FUNCTION_BLOCK BOXCOLOR_TO_COLOR (* Enum to Color *)
  (* Standard: 61499-2 *)
  (* Version 0.3, 2009-09-15, JHC, Holobloc Inc, Changed transition priorities. *)
  (* Version 0.2, 2003-12-04, JHC, Rockwell Automation, Renamed for better indexing. *)
  (* Version 0.1, 2002-11-05, JHC, Rockwell Automation, Corrected missing ST element in Algorithm REQ. *)
  (* Version 0.0, 2000-05-30, JHC, Rockwell Automation *)
  (* Compiler header: package fb.rt.dasdA1.A2.Box; *)
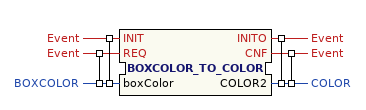
  EVENT_INPUT
    INIT WITH boxColor; (* Initialization Request *)
    REQ WITH boxColor; (* Normal Execution Request *)
  END_EVENT
  EVENT_OUTPUT
    INITO WITH COLOR2; (* Initialization Confirm *)
    CNF WITH COLOR2; (* Execution Confirmation *)
  END_EVENT
  VAR_INPUT
    boxColor : BOXCOLOR; (* BOXCOLOR ENUM *)
  END_VAR
  VAR_OUTPUT
    COLOR2 : COLOR; (* Color *)
  END_VAR
  VAR
    C2 : COLOR := COLOR#YELLOW;
    C3 : COLOR := COLOR#BLUE;
    C1 : COLOR := COLOR#RED;
  END_VAR
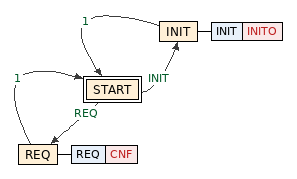
  EC_STATES
    START; (* Initial State *)
    INIT : INIT -> INITO; (* Initialization *)
    REQ : REQ -> CNF; (* Normal execution *)
  END_STATES
  EC_TRANSITIONS
    INIT TO START := 1;
    START TO REQ := REQ;
    START TO INIT := INIT;
    REQ TO START := 1;
  END_TRANSITIONS
  ALGORITHM INIT IN ST: (* Initialization algorithm *)

  END_ALGORITHM
  ALGORITHM REQ IN ST: (* Normally executed algorithm *)
IF (boxColor = BOXCOLOR.BLUE ) THEN
	COLOR2 := C3;
ELSIF (boxColor = BOXCOLOR.RED) THEN
	COLOR2 := C1;
ELSE
	COLOR2 := C2;
END_IF;
  END_ALGORITHM
END_FUNCTION_BLOCK
